// TwinCAT 3 PLC project TF6620_S7CommunicationSample_SysMan
// ProgramVersion: 3.1.4023.0
// libraries:
//   Tc2_Standard, * (Beckhoff Automation GmbH)
//   Tc2_System, * (Beckhoff Automation GmbH)
//   Tc3_Module, * (Beckhoff Automation GmbH)
// project tree:
//   DUTs/ ST_S7_Incoming.TcDUT, ST_S7_Incoming_Cyclic.TcDUT, ST_S7_Info.TcDUT, ST_S7_RequestHandling.TcDUT
//   / PlcTask.TcTTO
//   POUs/ MAIN.TcPOU
// real-time tasks:
//   TASK PlcTask: cycle T#10ms, priority 20, ADS port 350
// I/O:
//   DEVICE Device 1 (RT-Ethernet Adapter)
// variable links:
//   TF6620_S7CommunicationSample_SysMan/TF6620_S7CommunicationSample_SysMan Instance <-> Device 1 (RT-Ethernet Adapter)/Device 1 (RT-Ethernet Adapter)_Obj1 (TCP/UDP RT)/Object1 (S7 Connector)
//     PlcTask Inputs/MAIN.stS7Info.bS7Error <-> Status/Error
//     PlcTask Inputs/MAIN.stS7Info.eS7CommState <-> Status/State
//   TF6620_S7CommunicationSample_SysMan/TF6620_S7CommunicationSample_SysMan Instance <-> Device 1 (RT-Ethernet Adapter)/Device 1 (RT-Ethernet Adapter)_Obj1 (TCP/UDP RT)/Object1 (S7 Connector)/Object1 (S7 Single Request)
//     PlcTask Inputs/MAIN.stS7Incoming.b{1..4} <-> ReadFromS7/b{1..4}  (4 links)
//     PlcTask Inputs/MAIN.stS7Incoming.by1 <-> ReadFromS7/by1
//     PlcTask Inputs/MAIN.stS7Incoming.i1 <-> ReadFromS7/i1
//     PlcTask Inputs/MAIN.stS7Incoming.r1 <-> ReadFromS7/r1
//     PlcTask Inputs/MAIN.stS7Incoming.r2 <-> ReadFromS7/r2
//     PlcTask Inputs/MAIN.stS7Incoming.w1 <-> ReadFromS7/w1
//     PlcTask Inputs/MAIN.stS7RequestHandling.byReceiveCounter <-> Status/ReceiveCounter
//     PlcTask Outputs/MAIN.bWriteEnable <-> Control/WriteToS7Enable
//     PlcTask Outputs/MAIN.i1write <-> WriteToS7/i1
//     PlcTask Outputs/MAIN.stS7RequestHandling.bySendRequest <-> Control/SendRequest
//   TF6620_S7CommunicationSample_SysMan/TF6620_S7CommunicationSample_SysMan Instance <-> Device 1 (RT-Ethernet Adapter)/Device 1 (RT-Ethernet Adapter)_Obj1 (TCP/UDP RT)/Object1 (S7 Connector)/Object2 (S7 Cycle Request)
//     PlcTask Inputs/MAIN.stS7IncomingCyclic.b{1..4} <-> ReadFromS7/b{1..4}  (4 links)
//     PlcTask Inputs/MAIN.stS7IncomingCyclic.by1 <-> ReadFromS7/by1
//     PlcTask Inputs/MAIN.stS7IncomingCyclic.i1 <-> ReadFromS7/i1
//     PlcTask Inputs/MAIN.stS7IncomingCyclic.r1 <-> ReadFromS7/r1
//     PlcTask Inputs/MAIN.stS7IncomingCyclic.r2 <-> ReadFromS7/r2
//     PlcTask Inputs/MAIN.stS7IncomingCyclic.w1 <-> ReadFromS7/w1

CONFIGURATION TF6620_S7CommunicationSample_SysMan
    RESOURCE PLC ON TwinCAT3
        TASK PlcTask(INTERVAL := T#10ms, PRIORITY := 20);
        PROGRAM MAIN WITH PlcTask : MAIN;
    END_RESOURCE
END_CONFIGURATION

// ---- DUTs/ST_S7_Incoming.TcDUT
TYPE ST_S7_Incoming :
STRUCT
	by1 AT%I* 	: BYTE;
	b1 AT%I* 	: BOOL;
	b2 AT%I* 	: BOOL;
	b3 AT%I* 	: BOOL;
	b4 AT%I* 	: BOOL;
	w1 AT%I*	: DWORD;
	r1 AT%I*	: REAL;
	r2 AT%I*	: REAL;
	i1 AT%I*	: INT;	
END_STRUCT
END_TYPE

// ---- DUTs/ST_S7_Incoming_Cyclic.TcDUT
TYPE ST_S7_Incoming_Cyclic :
STRUCT
	by1 AT%I* 	: BYTE;
	b1 AT%I* 	: BOOL;
	b2 AT%I* 	: BOOL;
	b3 AT%I* 	: BOOL;
	b4 AT%I* 	: BOOL;
	w1 AT%I*	: DWORD;
	r1 AT%I*	: REAL;
	r2 AT%I*	: REAL;
	i1 AT%I*	: INT;	
END_STRUCT
END_TYPE

// ---- DUTs/ST_S7_Info.TcDUT
TYPE ST_S7_Info :
STRUCT
	eS7CommState AT%I* 	: BYTE;
	bS7Error AT%I* 		: BOOL;
END_STRUCT
END_TYPE

// ---- DUTs/ST_S7_RequestHandling.TcDUT
TYPE ST_S7_RequestHandling :
STRUCT
	bySendRequest AT%Q*		: BYTE;
	byReceiveCounter AT%I*	: BYTE;	
END_STRUCT
END_TYPE

// ---- POUs/MAIN.TcPOU
PROGRAM MAIN
VAR
	bStartReadRequest 	: BOOL;	
	bStartWriteRequest	: BOOL;
	
	stS7Info			: ST_S7_Info;
	stS7RequestHandling	: ST_S7_RequestHandling;

	(* Read variables *)
	bReadRequestDone	: BOOL;
	stS7Incoming		: ST_S7_Incoming;
	stS7IncomingCyclic	: ST_S7_Incoming_Cyclic;
	
	(* Write variables *)
	bWriteEnable AT%Q*	: BOOL;
	bWriteRequestDone	: BOOL;
	i1write AT%Q*		: INT := 42;
	
	(* State machine variables *)
	nStateRead			: UINT;
	nStateWrite			: UINT;
	
END_VAR

CASE nStateRead OF 
	
	// WAIT FOR START READ
	0: 
		IF bStartReadRequest THEN
			bStartReadRequest := FALSE;
			bReadRequestDone := FALSE;
			nStateRead := nStateRead + 1;
		END_IF

	// TRIGGER READ
	1:
		stS7RequestHandling.bySendRequest := stS7RequestHandling.byReceiveCounter + 1;
		nStateRead := nStateRead + 1;
		
	// WAIT FOR READ DONE
	2: 
		IF stS7RequestHandling.byReceiveCounter = stS7RequestHandling.bySendRequest THEN
			nStateRead := nStateRead + 1;
		END_IF	
		
	// DONE
	3: 
		bReadRequestDone := TRUE;
		nStateRead := 0;
	
END_CASE


CASE nStateWrite OF
	
	// WAIT FOR START WRITE
	0:
		IF bStartWriteRequest THEN
			bStartWriteRequest := FALSE;
			bWriteRequestDone := FALSE;
			bWriteEnable := TRUE;
			nStateWrite := nStateWrite + 1;
		END_IF

	// TRIGGER WRITE
	1:
		stS7RequestHandling.bySendRequest := stS7RequestHandling.byReceiveCounter + 1;
		nStateWrite := nStateWrite + 1;
		
	// WAIT FOR WRITE DONE
	2: 
		IF stS7RequestHandling.byReceiveCounter = stS7RequestHandling.bySendRequest THEN
			bWriteEnable := FALSE;
			nStateWrite := nStateWrite + 1;
		END_IF	
		
	// DONE
	3: 
		bWriteRequestDone := TRUE;
		nStateWrite := 0;
		
END_CASE

END_PROGRAM
